// TIA Portal V16 export
// export: Created 2022-02-04T14:40:10.4461478Z, ExportSetting WithDefaults, DisplayName Totally Integrated Automation Portal, DisplayVersion V16 Update 1, DisplayName TIA Portal Version Control Interface, DisplayVersion V16, DisplayName TIA Portal Openness, DisplayVersion V16, DisplayName SINAMICS Startdrive Advanced, DisplayVersion V16 Update 5, DisplayName SINAMICS Startdrive G130, G150, S120, S150, SINAMICS MV, S210, DisplayVersion V16 Update 5, DisplayName SINAMICS Startdrive G110M, G120, G120C, G120D, G120P, G115D, DisplayVersion V16 Update 5, DisplayName STEP 7 Professional, DisplayVersion V16, DisplayName STEP 7 Safety, DisplayVersion V16, DisplayName WinCC Advanced, DisplayVersion V16, DisplayName SIMATIC Visualization Architect, DisplayVersion V16
FUNCTION_BLOCK "Подача прокладки"   // FB6, LAD
VERSION : 0.1
// Подача прокладки
// stored: AutoNumber true, IsIECCheckEnabled false, UDAEnableTagReadback false
   VAR DB_SPECIFIC
      "TrigS84.4/S79.1" : Bool;
      Trig315 : Bool;
   END_VAR
   VAR_TEMP   // added for the SCL form of the ladder/FBD networks
      _w1 : Bool;
      _s5time1 : S5Time;
      _w2 : Bool;
      _w3 : Bool;
      _s5time2 : S5Time;
   END_VAR
BEGIN

REGION Network 1: Готовность
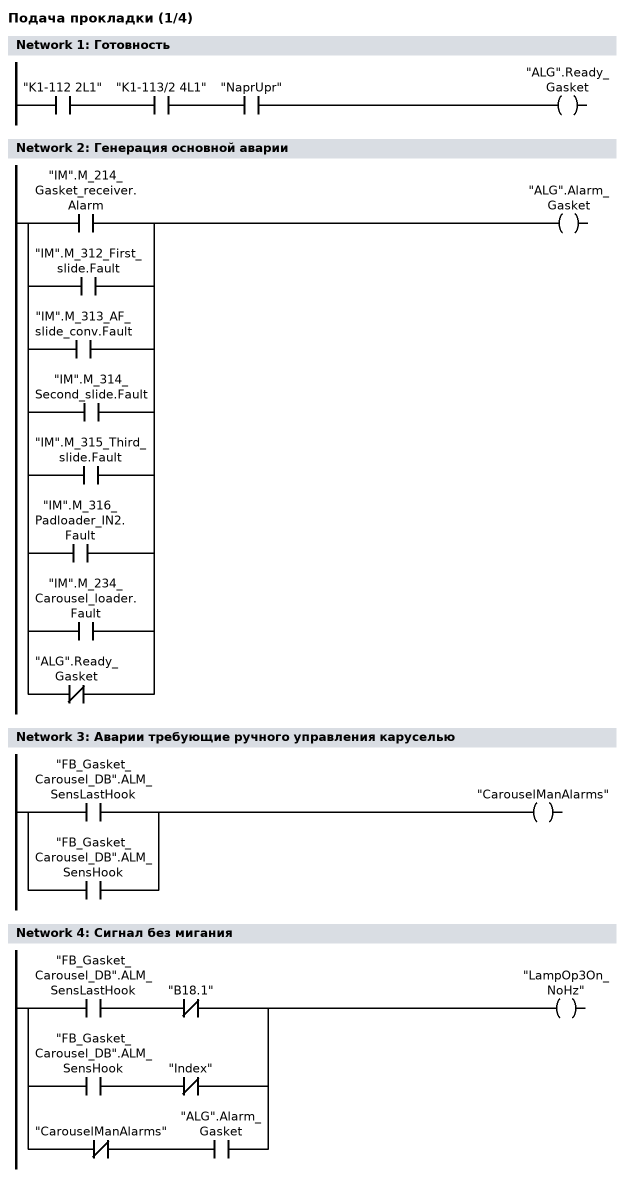
   RUNG wire#powerrail
      Contact( "K1-112 2L1" )
      Contact( "K1-113/2 4L1" )
      Contact( "NaprUpr" )
      Coil( "ALG".Ready_Gasket )
   END_RUNG
   // the same network as SCL:
   "ALG".Ready_Gasket := "K1-112 2L1" AND "K1-113/2 4L1" AND "NaprUpr";
END_REGION

REGION Network 2: Генерация основной аварии
   RUNG wire#powerrail
      Contact( "IM".M_214_Gasket_receiver.Alarm )
      wire#w1
      Coil( "ALG".Alarm_Gasket )
   END_RUNG
   RUNG wire#powerrail
      Contact( "IM".M_312_First_slide.Fault )
   END_RUNG wire#w1
   RUNG wire#powerrail
      Contact( "IM".M_313_AF_slide_conv.Fault )
   END_RUNG wire#w1
   RUNG wire#powerrail
      Contact( "IM".M_314_Second_slide.Fault )
   END_RUNG wire#w1
   RUNG wire#powerrail
      Contact( "IM".M_315_Third_slide.Fault )
   END_RUNG wire#w1
   RUNG wire#powerrail
      Contact( "IM".M_316_Padloader_IN2.Fault )
   END_RUNG wire#w1
   RUNG wire#powerrail
      Contact( "IM".M_234_Carousel_loader.Fault )
   END_RUNG wire#w1
   RUNG wire#powerrail
      I_Contact( "ALG".Ready_Gasket )
   END_RUNG wire#w1
   // the same network as SCL:
   "ALG".Alarm_Gasket := "IM".M_214_Gasket_receiver.Alarm OR "IM".M_312_First_slide.Fault OR "IM".M_313_AF_slide_conv.Fault OR "IM".M_314_Second_slide.Fault OR "IM".M_315_Third_slide.Fault OR "IM".M_316_Padloader_IN2.Fault OR "IM".M_234_Carousel_loader.Fault OR NOT "ALG".Ready_Gasket;
END_REGION

REGION Network 3: Аварии требующие ручного управления каруселью
   RUNG wire#powerrail
      Contact( "FB_Gasket_Carousel_DB".ALM_SensLastHook )
      wire#w1
      Coil( "CarouselManAlarms" )
   END_RUNG
   RUNG wire#powerrail
      Contact( "FB_Gasket_Carousel_DB".ALM_SensHook )
   END_RUNG wire#w1
   // the same network as SCL:
   "CarouselManAlarms" := "FB_Gasket_Carousel_DB".ALM_SensLastHook OR "FB_Gasket_Carousel_DB".ALM_SensHook;
END_REGION

REGION Network 4: Сигнал без мигания
   RUNG wire#powerrail
      Contact( "FB_Gasket_Carousel_DB".ALM_SensLastHook )
      I_Contact( "B18.1" )
      wire#w1
      Coil( "LampOp3On_NoHz" )
   END_RUNG
   RUNG wire#powerrail
      Contact( "FB_Gasket_Carousel_DB".ALM_SensHook )
      I_Contact( "Index" )
   END_RUNG wire#w1
   RUNG wire#powerrail
      I_Contact( "CarouselManAlarms" )
      Contact( "ALG".Alarm_Gasket )
   END_RUNG wire#w1
   // the same network as SCL:
   "LampOp3On_NoHz" := ("FB_Gasket_Carousel_DB".ALM_SensLastHook AND NOT "B18.1") OR ("FB_Gasket_Carousel_DB".ALM_SensHook AND NOT "Index") OR (NOT "CarouselManAlarms" AND "ALG".Alarm_Gasket);
END_REGION

REGION Network 5: Сигнал об авариях с миганием
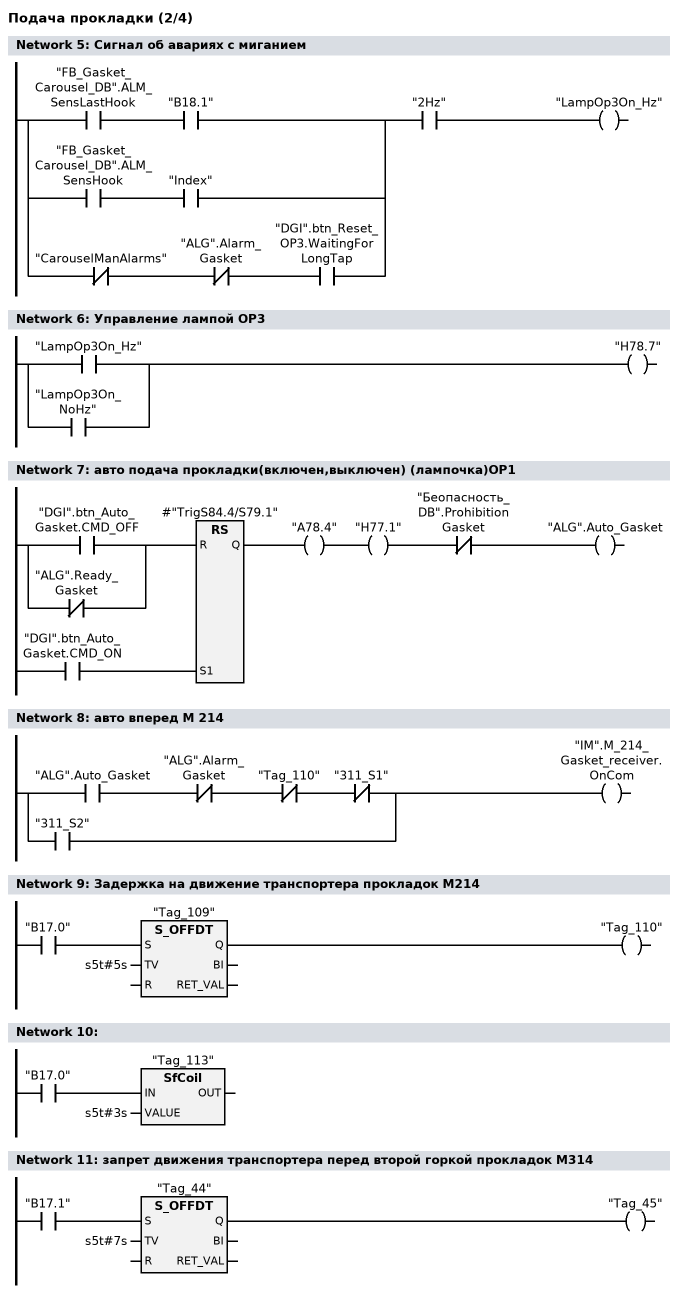
   RUNG wire#powerrail
      Contact( "FB_Gasket_Carousel_DB".ALM_SensLastHook )
      Contact( "B18.1" )
      wire#w1
      Contact( "2Hz" )
      Coil( "LampOp3On_Hz" )
   END_RUNG
   RUNG wire#powerrail
      Contact( "FB_Gasket_Carousel_DB".ALM_SensHook )
      Contact( "Index" )
   END_RUNG wire#w1
   RUNG wire#powerrail
      I_Contact( "CarouselManAlarms" )
      I_Contact( "ALG".Alarm_Gasket )
      Contact( "DGI".btn_Reset_OP3.WaitingForLongTap )
   END_RUNG wire#w1
   // the same network as SCL:
   "LampOp3On_Hz" := (("FB_Gasket_Carousel_DB".ALM_SensLastHook AND "B18.1") OR ("FB_Gasket_Carousel_DB".ALM_SensHook AND "Index") OR (NOT "CarouselManAlarms" AND NOT "ALG".Alarm_Gasket AND "DGI".btn_Reset_OP3.WaitingForLongTap)) AND "2Hz";
END_REGION

REGION Network 6: Управление лампой OP3
   RUNG wire#powerrail
      Contact( "LampOp3On_Hz" )
      wire#w1
      Coil( "H78.7" )
   END_RUNG
   RUNG wire#powerrail
      Contact( "LampOp3On_NoHz" )
   END_RUNG wire#w1
   // the same network as SCL:
   "H78.7" := "LampOp3On_Hz" OR "LampOp3On_NoHz";
END_REGION

REGION Network 7: авто подача прокладки(включен,выключен) (лампочка)ОР1
   RUNG wire#powerrail
      Contact( "DGI".btn_Auto_Gasket.CMD_OFF )
      wire#w1
      S_RS(operand := #"TrigS84.4/S79.1", s1 := wire#w2)
      Coil( "A78.4" )
      Coil( "H77.1" )
      I_Contact( "Беопасность_DB".ProhibitionGasket )
      Coil( "ALG".Auto_Gasket )
   END_RUNG
   RUNG wire#powerrail
      I_Contact( "ALG".Ready_Gasket )
   END_RUNG wire#w1
   RUNG wire#powerrail
      Contact( "DGI".btn_Auto_Gasket.CMD_ON )
   END_RUNG wire#w2
   // the same network as SCL:
   IF "DGI".btn_Auto_Gasket.CMD_OFF OR NOT "ALG".Ready_Gasket THEN
       #"TrigS84.4/S79.1" := FALSE;   // RS flip-flop
   END_IF;
   IF "DGI".btn_Auto_Gasket.CMD_ON THEN #"TrigS84.4/S79.1" := TRUE; END_IF;
   "A78.4" := #"TrigS84.4/S79.1";
   "H77.1" := #"TrigS84.4/S79.1";
   "ALG".Auto_Gasket := #"TrigS84.4/S79.1" AND NOT "Беопасность_DB".ProhibitionGasket;
END_REGION

REGION Network 8: авто вперед M 214
   RUNG wire#powerrail
      Contact( "ALG".Auto_Gasket )
      I_Contact( "ALG".Alarm_Gasket )
      I_Contact( "Tag_110" )
      I_Contact( "311_S1" )
      wire#w1
      Coil( "IM".M_214_Gasket_receiver.OnCom )
   END_RUNG
   RUNG wire#powerrail
      Contact( "311_S2" )
   END_RUNG wire#w1
   // the same network as SCL:
   "IM".M_214_Gasket_receiver.OnCom := ("ALG".Auto_Gasket AND NOT "ALG".Alarm_Gasket AND NOT "Tag_110" AND NOT "311_S1") OR "311_S2";
END_REGION

REGION Network 9: Задержка на движение транспортера прокладок М214
   RUNG wire#powerrail
      Contact( "B17.0" )
      S_OFFDT(T_NO := "Tag_109", TV := s5t#5s, R :=, BI =>, RET_VAL =>)
      Coil( "Tag_110" )
   END_RUNG
   // the same network as SCL:
   #_s5time1 := S_OFFDT(T_NO := "Tag_109", S := "B17.0", TV := s5t#5s, Q => #_w1);
   "Tag_110" := #_w1;
END_REGION

REGION Network 10
   // no SCL statement known for SfCoil: written as a call
   SfCoil(in := "B17.0", value := s5t#3s, operand := "Tag_113");
END_REGION

REGION Network 11: запрет движения транспортера перед второй горкой прокладок М314
   RUNG wire#powerrail
      Contact( "B17.1" )
      S_OFFDT(T_NO := "Tag_44", TV := s5t#7s, R :=, BI =>, RET_VAL =>)
      Coil( "Tag_45" )
   END_RUNG
   // the same network as SCL:
   #_s5time1 := S_OFFDT(T_NO := "Tag_44", S := "B17.1", TV := s5t#7s, Q => #_w1);
   "Tag_45" := #_w1;
END_REGION

REGION Network 12: Авто вперед команда подачи прокладок до горок
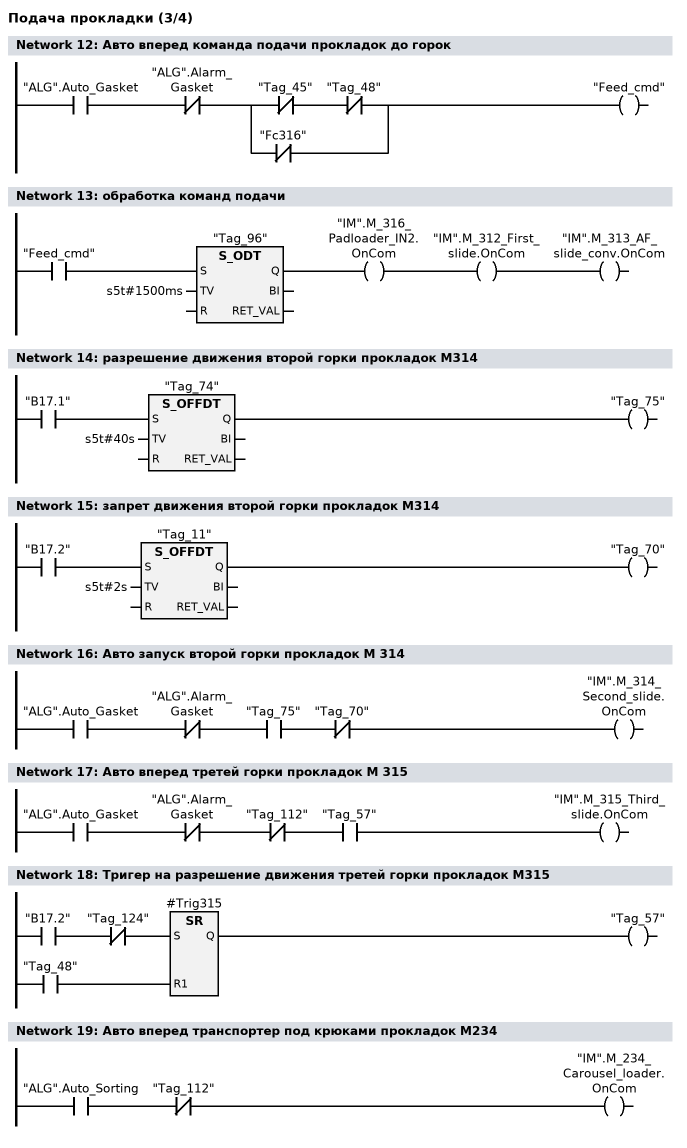
   RUNG wire#powerrail
      Contact( "ALG".Auto_Gasket )
      I_Contact( "ALG".Alarm_Gasket )
      wire#w1
      I_Contact( "Tag_45" )
      I_Contact( "Tag_48" )
      wire#w2
      Coil( "Feed_cmd" )
   END_RUNG
   RUNG wire#w1
      I_Contact( "Fc316" )
   END_RUNG wire#w2
   // the same network as SCL:
   "Feed_cmd" := "ALG".Auto_Gasket AND NOT "ALG".Alarm_Gasket AND ((NOT "Tag_45" AND NOT "Tag_48") OR NOT "Fc316");
END_REGION

REGION Network 13: обработка команд подачи
   RUNG wire#powerrail
      Contact( "Feed_cmd" )
      S_ODT(T_NO := "Tag_96", TV := s5t#1500ms, R :=, BI =>, RET_VAL =>)
      Coil( "IM".M_316_Padloader_IN2.OnCom )
      Coil( "IM".M_312_First_slide.OnCom )
      Coil( "IM".M_313_AF_slide_conv.OnCom )
   END_RUNG
   // the same network as SCL:
   #_s5time1 := S_ODT(T_NO := "Tag_96", S := "Feed_cmd", TV := s5t#1500ms, Q => #_w1);
   "IM".M_316_Padloader_IN2.OnCom := #_w1;
   "IM".M_312_First_slide.OnCom := #_w1;
   "IM".M_313_AF_slide_conv.OnCom := #_w1;
END_REGION

REGION Network 14: разрешение движения второй горки прокладок М314
   RUNG wire#powerrail
      Contact( "B17.1" )
      S_OFFDT(T_NO := "Tag_74", TV := s5t#40s, R :=, BI =>, RET_VAL =>)
      Coil( "Tag_75" )
   END_RUNG
   // the same network as SCL:
   #_s5time1 := S_OFFDT(T_NO := "Tag_74", S := "B17.1", TV := s5t#40s, Q => #_w1);
   "Tag_75" := #_w1;
END_REGION

REGION Network 15: запрет движения второй горки прокладок М314
   RUNG wire#powerrail
      Contact( "B17.2" )
      S_OFFDT(T_NO := "Tag_11", TV := s5t#2s, R :=, BI =>, RET_VAL =>)
      Coil( "Tag_70" )
   END_RUNG
   // the same network as SCL:
   #_s5time1 := S_OFFDT(T_NO := "Tag_11", S := "B17.2", TV := s5t#2s, Q => #_w1);
   "Tag_70" := #_w1;
END_REGION

REGION Network 16: Авто запуск второй горки прокладок М 314
   RUNG wire#powerrail
      Contact( "ALG".Auto_Gasket )
      I_Contact( "ALG".Alarm_Gasket )
      Contact( "Tag_75" )
      I_Contact( "Tag_70" )
      Coil( "IM".M_314_Second_slide.OnCom )
   END_RUNG
   // the same network as SCL:
   "IM".M_314_Second_slide.OnCom := "ALG".Auto_Gasket AND NOT "ALG".Alarm_Gasket AND "Tag_75" AND NOT "Tag_70";
END_REGION

REGION Network 17: Авто вперед третей горки прокладок M 315
   RUNG wire#powerrail
      Contact( "ALG".Auto_Gasket )
      I_Contact( "ALG".Alarm_Gasket )
      I_Contact( "Tag_112" )
      Contact( "Tag_57" )
      Coil( "IM".M_315_Third_slide.OnCom )
   END_RUNG
   // the same network as SCL:
   "IM".M_315_Third_slide.OnCom := "ALG".Auto_Gasket AND NOT "ALG".Alarm_Gasket AND NOT "Tag_112" AND "Tag_57";
END_REGION

REGION Network 18: Тригер на разрешение движения третей горки прокладок М315
   RUNG wire#powerrail
      Contact( "B17.2" )
      I_Contact( "Tag_124" )
      S_SR(operand := #Trig315, r1 := wire#w1)
      Coil( "Tag_57" )
   END_RUNG
   RUNG wire#powerrail
      Contact( "Tag_48" )
   END_RUNG wire#w1
   // the same network as SCL:
   IF "B17.2" AND NOT "Tag_124" THEN
       #Trig315 := TRUE;   // SR flip-flop
   END_IF;
   IF "Tag_48" THEN #Trig315 := FALSE; END_IF;
   "Tag_57" := #Trig315;
END_REGION

REGION Network 19: Авто вперед транспортер под крюками прокладок M234
   RUNG wire#powerrail
      Contact( "ALG".Auto_Sorting )
      I_Contact( "Tag_112" )
      Coil( "IM".M_234_Carousel_loader.OnCom )
   END_RUNG
   // the same network as SCL:
   "IM".M_234_Carousel_loader.OnCom := "ALG".Auto_Sorting AND NOT "Tag_112";
END_REGION

REGION Network 20: Задержка на датчик максимального слоя прокладки 234.2
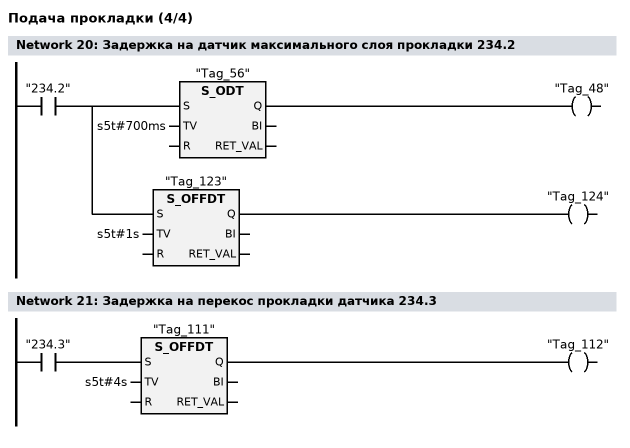
   RUNG wire#powerrail
      Contact( "234.2" )
      wire#w1
      S_ODT(T_NO := "Tag_56", TV := s5t#700ms, R :=, BI =>, RET_VAL =>)
      Coil( "Tag_48" )
   END_RUNG
   RUNG wire#w1
      S_OFFDT(T_NO := "Tag_123", TV := s5t#1s, R :=, BI =>, RET_VAL =>)
      Coil( "Tag_124" )
   END_RUNG
   // the same network as SCL:
   #_w2 := "234.2";
   #_s5time1 := S_ODT(T_NO := "Tag_56", S := "234.2", TV := s5t#700ms, Q => #_w1);
   "Tag_48" := #_w1;
   #_s5time2 := S_OFFDT(T_NO := "Tag_123", S := #_w2, TV := s5t#1s, Q => #_w3);
   "Tag_124" := #_w3;
END_REGION

REGION Network 21: Задержка на перекос прокладки датчика 234.3
   RUNG wire#powerrail
      Contact( "234.3" )
      S_OFFDT(T_NO := "Tag_111", TV := s5t#4s, R :=, BI =>, RET_VAL =>)
      Coil( "Tag_112" )
   END_RUNG
   // the same network as SCL:
   #_s5time1 := S_OFFDT(T_NO := "Tag_111", S := "234.3", TV := s5t#4s, Q => #_w1);
   "Tag_112" := #_w1;
END_REGION
END_FUNCTION_BLOCK
